(*

.. <legal notes>

legal notes
=================
| SPDX-FileCopyrightText: © 2026 Oleksandr Tiutyk <trofimich@gmail.com>
| SPDX-License-Identifier: LGPL-3.0-only
| For details check: LGPL-3.0-only_

.. _LGPL-3.0-only: https://www.gnu.org/licenses/lgpl-3.0.en.html

.. </legal notes>

*)

PROGRAM RealHelper
VAR CONSTANT
	MIN_VALUE : REAL := -3.402823E+38;
	MAX_VALUE : REAL := +3.402823E+38;
END_VAR
VAR
	_ClassName : STRING := __POUNAME();
END_VAR

{attribute 'monitoring' := 'call'}
PROPERTY ClassName : STRING
GET
ClassName := _ClassName;
END_GET
END_PROPERTY

{attribute 'monitoring' := 'call'}
PROPERTY NamespaceName : STRING
GET
NamespaceName := CurrentNamespace.Name;
END_GET
END_PROPERTY

END_PROGRAM

(* stored: Version 1.1.0.1
   POU RealHelper: Id {361c062a-943b-4db7-ab4a-7715ff446a31}, SpecialFunc None
   Property ClassName: Id {9df65ee2-61ad-4aa6-8540-da6369d277dd}
   Get Get: Id {f3e499ff-278e-4944-9b5a-c3c32eaeeaeb}
   Property NamespaceName: Id {38bfc198-2daa-457d-8569-d0dd6eafc0d0}
   Get Get: Id {f423181e-b835-486d-a0e9-cbf1e9bf75ba} *)
